FUNCTION_BLOCK PID
  (* Standard: 61499-2 *)
  (* Version 0.1, 2017-00-02, hpea485, UOA *)
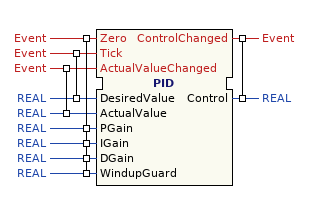
  EVENT_INPUT
    Zero WITH PGain, IGain, DGain, WindupGuard;
    Tick WITH DesiredValue;
    ActualValueChanged WITH ActualValue;
  END_EVENT
  EVENT_OUTPUT
    ControlChanged WITH Control;
  END_EVENT
  VAR_INPUT
    DesiredValue : REAL;
    ActualValue : REAL;
    PGain : REAL;
    IGain : REAL;
    DGain : REAL;
    WindupGuard : REAL;
  END_VAR
  VAR_OUTPUT
    Control : REAL;
  END_VAR
  VAR
    PreviousError : REAL;
    IntegrationError : REAL;
  END_VAR
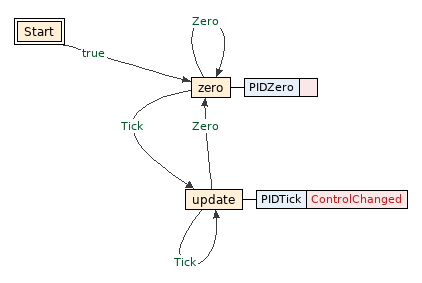
  EC_STATES
    Start;
    update : PIDTick -> ControlChanged;
    zero : PIDZero;
  END_STATES
  EC_TRANSITIONS
    Start TO zero := true;
    update TO zero := Zero;
    update TO update := Tick;
    zero TO update := Tick;
    zero TO zero := Zero;
  END_TRANSITIONS
  ALGORITHM PIDTick IN C:
	REAL diff;
	REAL p_term;
	REAL i_term;
	REAL d_term;

	REAL currentError = me->DesiredValue - me->ActualValue;

    // integration with windup guarding
    me->IntegrationError += currentError;
    if (me->IntegrationError < -(me->WindupGuard)) {
        me->IntegrationError = -(me->WindupGuard);

	} else if (me->IntegrationError > me->WindupGuard) {
        me->IntegrationError = me->WindupGuard;

	}

    // differentiation
    diff = currentError - me->PreviousError;

    // scaling
    p_term = (me->PGain * currentError);
    i_term = (me->IGain * me->IntegrationError);
    d_term = (me->DGain * diff);

    // summation of terms
    me->Control = p_term + i_term + d_term;

    // save current error as previous error for next iteration
    me->PreviousError = currentError;
  END_ALGORITHM
  ALGORITHM PIDZero IN C:
me->PreviousError = 0.0;
me->IntegrationError = 0.0;
  END_ALGORITHM
END_FUNCTION_BLOCK
